# EPICS substitutions: ek9000App/Db/EL2002.substitutions
file EL2002.template
{ 	pattern
	{
		TERMINAL,
		DESC1,	ZNAM1,	ONAM1,	PINI1,
		DESC2,	ZNAM2,	ONAM2,	PINI2
	}
	{
	}
}
